PROGRAM Vision_StateMachine
VAR
//var to get struct data from ck_real_value function
cx_vision_data : ck_real_flag_data;
cy_vision_data : ck_real_flag_data;
nut_turn_data : ck_real_flag_data;

sep_pos_data : ck_real_flag_data;

sep_rot_rigth_data :ck_real_flag_data;
sep_rot_left_data :ck_real_flag_data;
END_VAR

VAR_INPUT
		
init_: BOOL:= FALSE;
G_STATE: INT:=-1;
	
END_VAR


VAR RETAIN    
   
	Act_Gl_State :INT:=-1;
	Act_In_State: INT:=-1;
	
END_VAR


VAR CONSTANT 
	SeparatorPos:INT := 10;
	SeparatorPos_I:INT := 100;
	SeparatorPos_F:INT := 101;
	
	SeparatorRot:INT:= 11;
	SeparatorRot_I:INT:= 110;
	SeparatorRot_F:INT:= 111;
	
	SeparatorNut:INT:=12;
	SeparatorNut_I:INT:=120;
	SeparatorNut_F:INT:=121;
	
END_VAR

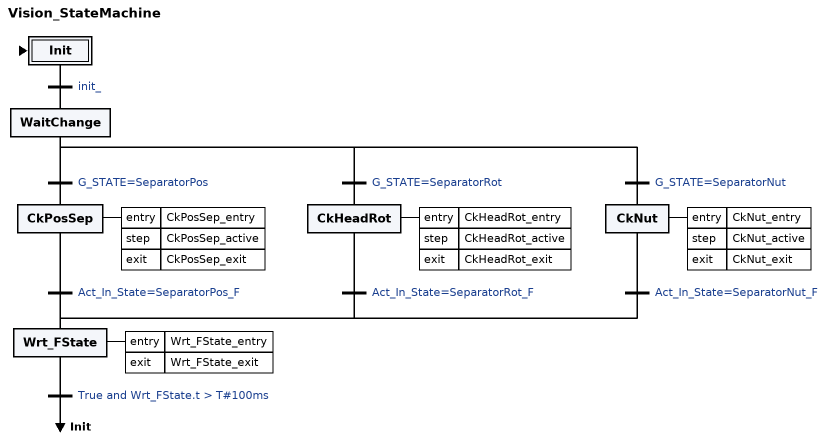
INITIAL_STEP Init:
END_STEP
TRANSITION FROM Init TO WaitChange
    := init_;
END_TRANSITION
STEP WaitChange:
END_STEP
TRANSITION FROM WaitChange TO CkPosSep
    := G_STATE=SeparatorPos;
END_TRANSITION
STEP CkPosSep:
    CkPosSep_entry(P1);  // entry action
    CkPosSep_active(N);  // step action
    CkPosSep_exit(P0);  // exit action
END_STEP
TRANSITION FROM CkPosSep TO Wrt_FState
    := Act_In_State=SeparatorPos_F;
END_TRANSITION
TRANSITION FROM WaitChange TO CkHeadRot
    := G_STATE=SeparatorRot;
END_TRANSITION
STEP CkHeadRot:
    CkHeadRot_entry(P1);  // entry action
    CkHeadRot_active(N);  // step action
    CkHeadRot_exit(P0);  // exit action
END_STEP
TRANSITION FROM CkHeadRot TO Wrt_FState
    := Act_In_State=SeparatorRot_F;
END_TRANSITION
TRANSITION FROM WaitChange TO CkNut
    := G_STATE=SeparatorNut;
END_TRANSITION
STEP CkNut:
    CkNut_entry(P1);  // entry action
    CkNut_active(N);  // step action
    CkNut_exit(P0);  // exit action
END_STEP
TRANSITION FROM CkNut TO Wrt_FState
    := Act_In_State=SeparatorNut_F;
END_TRANSITION
STEP Wrt_FState:
    Wrt_FState_entry(P1);  // entry action
    Wrt_FState_exit(P0);  // exit action
END_STEP
TRANSITION FROM Wrt_FState TO Init
    := True and Wrt_FState.t > T#100ms;
END_TRANSITION

ACTION CkHeadRot_active:
//verifies that the vision system has completed its task
IF ck_bool_value(Vision_struct.Ck_finish_procees) THEN 
	//read the values processed by the vision system and send to robot
	sep_rot_rigth_data := ck_real_value(Vision_struct.Head_rigth_value);
	sep_rot_left_data := ck_real_value(Vision_struct.Head_left_value);
	//check if all values are correct
	IF sep_rot_rigth_data.Flag AND sep_rot_left_data.Flag THEN
		//write variables from PLC to CS.UR5 Robot
		IF wr_real_value(Vision_const.HEAD_RIGTH_VALUE,sep_rot_rigth_data.Value) THEN
			IF wr_real_value(Vision_const.HEAD_LEFT_VALUE,sep_rot_left_data.Value) THEN
					//change the value of variable
					Vision_struct.Ck_finish_procees.Flag1:=FALSE;
					Vision_struct.Ck_finish_procees.Flag2:=FALSE;
					Vision_struct.Ck_finish_procees.Flag3:=FALSE;			
					Act_In_State := SeparatorRot_F;
			END_IF

			  END_IF
		END_IF
	END_IF
END_ACTION

ACTION CkHeadRot_entry:


//write the retain state variable 
Act_Gl_State:=SeparatorRot;

//start the vision system
Vision_struct.Get_img_head_left_rot.Flag1:=TRUE;
Vision_struct.Get_img_head_left_rot.Flag2:=TRUE;
Vision_struct.Get_img_head_left_rot.Flag3:=TRUE;

Vision_struct.Get_img_head_rigth_rot.Flag1:=TRUE;
Vision_struct.Get_img_head_rigth_rot.Flag2:=TRUE;
Vision_struct.Get_img_head_rigth_rot.Flag3:=TRUE;

Act_In_State := SeparatorRot_I;
END_ACTION

ACTION CkHeadRot_exit:
//write reset state variables to robot.
//wr_state(CS.UR5,RESET_STATE);
//reset Global state variable
G_STATE := -1;

//reset the vision system
Vision_struct.Get_img_head_left_rot.Flag1:=FALSE;
Vision_struct.Get_img_head_left_rot.Flag2:=FALSE;
Vision_struct.Get_img_head_left_rot.Flag3:=FALSE;

Vision_struct.Get_img_head_rigth_rot.Flag1:=FALSE;
Vision_struct.Get_img_head_rigth_rot.Flag2:=FALSE;
Vision_struct.Get_img_head_rigth_rot.Flag3:=FALSE;
END_ACTION

ACTION CkNut_active:
//verifies that the vision system has completed its task
IF ck_bool_value(Vision_struct.Ck_finish_procees) THEN 
	//read the values processed by the vision system and send to robot
	cx_vision_data := ck_real_value(Vision_struct.Cx_value);
	cy_vision_data := ck_real_value(Vision_struct.Cy_value);
	nut_turn_data := ck_real_value(Vision_struct.Nut_turn_value);
	
	//check if all values are correct
	IF cx_vision_data.Flag AND cy_vision_data.Flag AND nut_turn_data.Flag THEN
		//write variables from PLC to CS.UR5 Robot
		IF wr_real_value(Vision_const.CX_VALUE,cx_vision_data.Value) THEN
			IF wr_real_value(Vision_const.CY_VALUE,cy_vision_data.Value) THEN
			  IF wr_real_value(Vision_const.NUT_VALUE,nut_turn_data.Value) THEN
					//change the value of variable
					Vision_struct.Ck_finish_procees.Flag1:=FALSE;
					Vision_struct.Ck_finish_procees.Flag1:=FALSE;
					Vision_struct.Ck_finish_procees.Flag1:=FALSE;
					Act_In_State := SeparatorNut_F;
			  END_IF
		END_IF
	END_IF
	END_IF
END_IF
END_ACTION

ACTION CkNut_entry:


//write the retain state variable 
Act_Gl_State:=SeparatorNut;

//start the vision system
Vision_struct.Get_img_nut.Flag1:= FALSE;
Vision_struct.Get_img_nut.Flag2:= FALSE;
Vision_struct.Get_img_nut.Flag3:= FALSE;

Act_In_State := SeparatorNut_I;
END_ACTION

ACTION CkNut_exit:
//reset Global state variable
G_STATE := -1;

//start the vision system
Vision_struct.Get_img_nut.Flag1:= TRUE;
Vision_struct.Get_img_nut.Flag2:= TRUE;
Vision_struct.Get_img_nut.Flag3:= TRUE;
END_ACTION

ACTION CkPosSep_active:
//verifies that the vision system has completed its task
IF ck_bool_value(Vision_struct.Ck_finish_procees) THEN 
	//read the values processed by the vision system and send to robot
	sep_pos_data := ck_real_value(Vision_struct.Pos_sep);
	//check if all values are correct
	IF sep_pos_data.Flag THEN
		//write variables from PLC to CS.UR5 Robot
		IF wr_real_value(Vision_const.SEP_POS_VALUE,sep_pos_data.Value) THEN
					//change the value of variable
					Vision_struct.Ck_finish_procees.Flag1:=FALSE;
					Vision_struct.Ck_finish_procees.Flag2:=FALSE;
					Vision_struct.Ck_finish_procees.Flag3:=FALSE;			
					Act_In_State := SeparatorPos_F;
			  END_IF
		END_IF
	END_IF
END_ACTION

ACTION CkPosSep_entry:


//write the retain state variable 
Act_Gl_State:=SeparatorPos;

//start the vision system
Vision_struct.Get_img_nut.Flag1:= TRUE;
Vision_struct.Get_img_nut.Flag2:= TRUE;
Vision_struct.Get_img_nut.Flag3:= TRUE;

Act_In_State := SeparatorPos_I;
END_ACTION

ACTION CkPosSep_exit:
//write reset state variables to robot.
//wr_state(CS.UR5,RESET_STATE);
//reset Global state variable
G_STATE := -1;



//Reset Vision varibles					
Vision_struct.Get_img_nut.Flag1:= TRUE;
Vision_struct.Get_img_nut.Flag2:= TRUE;
Vision_struct.Get_img_nut.Flag3:= TRUE;
END_ACTION

END_PROGRAM

(* stored: Version 1.1.0.1, ProductVersion 3.1.4024.4
   POU Vision_StateMachine: Id {f93bb11a-f5cd-40ad-a452-b50656e25a24}, SpecialFunc None
   Action CkHeadRot_active: Id {79483949-fdb1-43c7-85b0-66a3b8676161}
   Action CkHeadRot_entry: Id {7ebbfc85-5aad-4741-9c48-8a8ecd05823e}
   Action CkHeadRot_exit: Id {8e1964bb-4c65-4438-8d8b-94b34bd867af}
   Action CkNut_active: Id {a76c4aea-c03d-4f2e-a27c-e3588e7a8d51}
   Action CkNut_entry: Id {7b639d02-350f-49a2-9682-bc001a1885d5}
   Action CkNut_exit: Id {d8ded961-8fc2-4dab-9fb9-edf8d208d7d5}
   Action CkPosSep_active: Id {5eb9aaf2-ba77-4c72-8011-fd3d40ba003d}
   Action CkPosSep_entry: Id {90dd64f5-3a3d-4fd1-ac87-8dfd3a83d6a7}
   Action CkPosSep_exit: Id {b8d496af-bbe4-4811-b6ee-ef9fbec01c2f} *)
